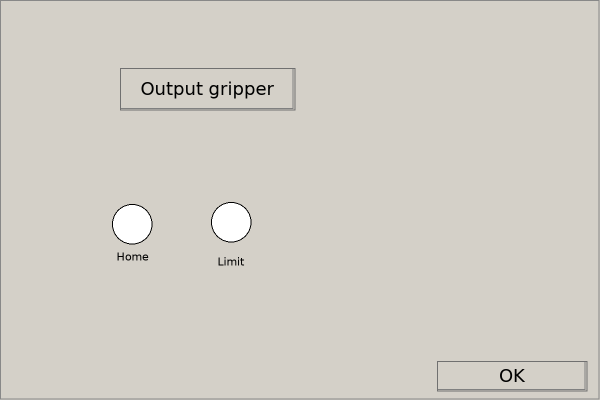
VISUALIZATION Dialog_Output  // 600x400
    Button (437,361 150x30), "OK"
        OnMouseClick: CloseDialog Dialog=Dialog_Output, Result=OK, NumpadKeypadSet=True
    Ellipse (112,204 40x40), colour toggle: gMachineCtrl.IO.In.HomeOutAxis
    Button (120,68 175x42), "Output gripper"
        toggle gMachineCtrl.IO.Out.Output_GripperClose
    Ellipse (211,202 40x40), colour toggle: gMachineCtrl.IO.In.HomeOutAxisLimit
    Label (102,242 62x30), "Home"
    Label (200,247 62x30), "Limit"
END_VISUALIZATION

(* stored: Version 1.1.0.1, ProductVersion 3.1.4024.3
   Visu Dialog_Output: Id {dfe65289-4455-46c7-897d-3a455ba1e590} *)
